TYPE "LubrValve_Wng"
VERSION : 0.1
// Block: LubrValve_Wng
   STRUCT
      SystemNotON : Bool;
   END_STRUCT;

END_TYPE
